// TIA Portal V19 export
TYPE "Thickness_PersData"
   STRUCT
      Measure { ExternalWritable := 'False'} : Struct
         BypassON : Bool;
         ID : DInt;   // Measurement Item Number
         Last_TriggerPosition : LReal;   // Previous Thickness Measurement
         AverageSum { ExternalAccessible := 'False'; ExternalVisible := 'False'} : LReal;   // Sum of Measurements for Average Calculation
         OutOfRange_Counter : Int;   // Number of out-of-range Thickness Measurements
         InRange_Counter : Int;   // Number of In-range Thickness Measurements
         Buffer : Array[1.."THICKNESS_CHECK__BUFFER_ITEMS"] of "Thickness_Measure_Item";   // Measurement Buffer Archive
      END_STRUCT;
      MES_Record { ExternalWritable := 'False'} : "Thickness_Measure_Item";
   END_STRUCT;
END_TYPE
